FUNCTION QUARTERS_TO_WORD
  (* Standard: 61499-1 *)
  (* Version 1.0, 2024-02-22, franz *)
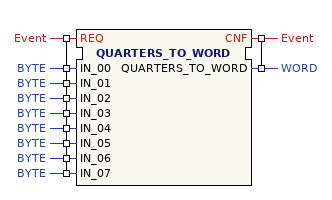
  EVENT_INPUT
    REQ WITH IN_00, IN_01, IN_02, IN_03, IN_04, IN_05, IN_06, IN_07;
  END_EVENT
  EVENT_OUTPUT
    CNF WITH QUARTERS_TO_WORD;
  END_EVENT
  VAR_INPUT
    IN_00 : BYTE; (* QUARTER BYTE 00 *)
    IN_01 : BYTE; (* QUARTER BYTE 01 *)
    IN_02 : BYTE; (* QUARTER BYTE 02 *)
    IN_03 : BYTE; (* QUARTER BYTE 03 *)
    IN_04 : BYTE; (* QUARTER BYTE 04 *)
    IN_05 : BYTE; (* QUARTER BYTE 05 *)
    IN_06 : BYTE; (* QUARTER BYTE 06 *)
    IN_07 : BYTE; (* QUARTER BYTE 07 *)
  END_VAR
  VAR_OUTPUT
    QUARTERS_TO_WORD : WORD;
  END_VAR
  BODY IN ST:
FUNCTION QUARTERS_TO_WORD : WORD

VAR_INPUT
	IN_00 : BYTE;    // QUARTER BYTE 00
	IN_01 : BYTE;    // QUARTER BYTE 01
	IN_02 : BYTE;    // QUARTER BYTE 02
	IN_03 : BYTE;    // QUARTER BYTE 03
	IN_04 : BYTE;    // QUARTER BYTE 04
	IN_05 : BYTE;    // QUARTER BYTE 05
	IN_06 : BYTE;    // QUARTER BYTE 06
	IN_07 : BYTE;    // QUARTER BYTE 07
END_VAR

(* this Function combines the 8 QUARTER BYTES to a word *)
QUARTERS_TO_WORD := WORD_QUARTER_ZZ;
QUARTERS_TO_WORD := QUARTERS_TO_WORD OR SHL(BYTE_TO_WORD(IN_07), SHFT_QUARTER_07);
QUARTERS_TO_WORD := QUARTERS_TO_WORD OR SHL(BYTE_TO_WORD(IN_06), SHFT_QUARTER_06);
QUARTERS_TO_WORD := QUARTERS_TO_WORD OR SHL(BYTE_TO_WORD(IN_05), SHFT_QUARTER_05);
QUARTERS_TO_WORD := QUARTERS_TO_WORD OR SHL(BYTE_TO_WORD(IN_04), SHFT_QUARTER_04);
QUARTERS_TO_WORD := QUARTERS_TO_WORD OR SHL(BYTE_TO_WORD(IN_03), SHFT_QUARTER_03);
QUARTERS_TO_WORD := QUARTERS_TO_WORD OR SHL(BYTE_TO_WORD(IN_02), SHFT_QUARTER_02);
QUARTERS_TO_WORD := QUARTERS_TO_WORD OR SHL(BYTE_TO_WORD(IN_01), SHFT_QUARTER_01);
QUARTERS_TO_WORD := QUARTERS_TO_WORD OR SHL(BYTE_TO_WORD(IN_00), SHFT_QUARTER_00);

END_FUNCTION
  END_BODY
END_FUNCTION
